{attribute 'qualified_only'}
{attribute 'strict'}
TYPE enRecMan_ErrorList :
(
	NoError := 0,
	ReloadRecipeListError:= 1,
	WriteRecipeError := 2,
	ReadRecipeError := 3,
	WriteSizeError:= 4,
	ReadSizeError:= 5,
	StructToBig:= 6,
	FileOpenError:= 7,
	FileCloseError:= 8,
	ReadRecipeTimeout:= 9,
	WriteRecipeTimeout:= 10,
	BadCRC:= 11,
	CommandStartProgramError:=12,
	FileDeleteError:=13,
	DeleteRecipeTimeout := 14
);
END_TYPE

(* stored: Version 1.1.0.1, ProductVersion 3.1.4024.4
   EnumerationTextList enRecMan_ErrorList: Id {2cf0ff80-5124-469f-a0f3-4f5257e2cad0} *)
